FUNCTION_BLOCK TcoInputDialogContentContainer EXTENDS TcoObject

END_FUNCTION_BLOCK

(* stored: Version 1.1.0.1
   POU TcoInputDialogContentContainer: Id {90d00f9b-0142-0ac3-077b-97c780db421c}, SpecialFunc None *)
